FUNCTION_BLOCK CU040AutomatTask EXTENDS CUBaseAutomat IMPLEMENTS ICUTask
VAR

    _missingProcessSettingMessage : TcoCore.TcoMessenger(THIS^);
    _paralellTask : CU040AutomatParalell_1_Task(THIS^, TcoCore.eRestoreMode.None);
	
	//~
    _sb : TcoCore.StringBuilder;
	//~
    _customizedContentInput : CU040DialogContent(THIS^);
END_VAR

VAR
    _dataLoadProcessSettings : BOOL;
    _dataLoadProcessSettingsByPlaner : BOOL;
    _dataCreateNew : BOOL;
    _dataOpen : BOOL;
    _dataClose : BOOL;
    _dataFinalize : BOOL;
    _continueRestore : BOOL;
    _loop : BOOL;
    _inspectionResult : BOOL;
    _inspectionDimensionResult : REAL;
    _tagsPairing : BOOL;
    _reqKey : STRING;
    _reqAssignedValue : STRING;
    _inspectorSingleExamples : BOOL;
    _inspectorGroupExamples : BOOL;
	_dialogExamples : BOOL;

END_VAR

Run();

(*~
	<docu>
		<summary>
			Loads technology settings from the current technology set into this controlled unit.
			The `StationProcessDataManager.Data` is populated by data from process settings.						
		</summary>
	</docu>
~*)
METHOD DataLoadProcessSettings : BOOL
VAR_INPUT
	inStepID : INT;
END_VAR

VAR
	_ans: TcoCore.eDialogAnswer;
END_VAR
IF (Step(inStepID, _dataLoadProcessSettings, 'LOAD PROCESS SETTING')) THEN
    //-------------------------------------
	
	THIS^._missingProcessSettingMessage.OnCondition(Station.Technology.ProcessSettings.Data._EntityId = '')
									   .Build()
									   .Append('No process data. Please load setting')
									   .As()				   
									   .AsError()
									   .Pin();
					   
				   
	IF(Station.Technology.ProcessSettings.Data._EntityId <> '' (*AND NOT THIS^._missingProcessSettingMessage.Pinned*)) THEN
		IF(Station.Technology.ProcessSettings.Read(Station.Technology.ProcessSettings.Data._EntityId).Done) THEN
			Station.ProcessDataManager.Data := Station.Technology.ProcessSettings.Data;
			Station.ProcessDataManager.Data.EntityHeader.RecipeCreated := Station.Technology.ProcessSettings.Data._Created;
			Station.ProcessDataManager.Data.EntityHeader.RecipeLastModified  := Station.Technology.ProcessSettings.Data._Modified;
			Station.ProcessDataManager.Data.EntityHeader.Recipe  := Station.Technology.ProcessSettings.Data._EntityId;				
			CompleteStep();

		END_IF;	
	ELSE
		_ans:=_dialog.Show()
			.WithImage('d:\MTS\Develop\TcOpenGroup\TcOpen\assets\logo\TcOpenWide.png',400,600)	
	       .WithCaption('<#Process data not selected#>')
		   .WithText('<#Would you like to load default settings?#>')
		   .WithYesNoCancel().Answer;
		IF(_ans=TcoCore.eDialogAnswer.Cancel) THEN
			this^.Restore();
		END_IF
		IF( _ans= TcoCore.eDialogAnswer.Yes) THEN
		   
		   	Station.Technology.ProcessSettings.Data._EntityId := 'default';
		END_IF; 

			
	END_IF		    				
    //-------------------------------------
END_IF
END_METHOD

(*~
	<docu>
		<summary>
			Loads process settings from the current process set into this controlled unit.
			The `StationProcessDataManager.Data` is populated by data from process settings.						
		</summary>
	</docu>
~*)
METHOD DataLoadProcessSettingsByPlaner : BOOL
VAR_INPUT
	inStepID : INT;
END_VAR
IF (Step(inStepID, _dataLoadProcessSettingsByPlaner, 'LOAD PROCESS SETTING BY THE PRODUCTION PLANER')) THEN
    //-------------------------------------


								   
	 IF Station.ProductionPlanerTask.Invoke().Done	AND_THEN(Station.ProductionPlanerTask.RequiredProcessSettingsId <> '') THEN
		
		IF NOT Station.ProductionPlanerTask.ProductionPlanCompleted and_then (Station.Technology.ProcessSettings.Read(Station.ProductionPlanerTask.RequiredProcessSettingsId).Done)
			 THEN
			Station.ProcessDataManager.Data := Station.Technology.ProcessSettings.Data;
			Station.ProcessDataManager.Data.EntityHeader.RecipeCreated := Station.Technology.ProcessSettings.Data._Created;
			Station.ProcessDataManager.Data.EntityHeader.RecipeLastModified  := Station.Technology.ProcessSettings.Data._Modified;
			Station.ProcessDataManager.Data.EntityHeader.Recipe  := Station.Technology.ProcessSettings.Data._EntityId;				
			CompleteStep();
			Station.ProductionPlanerTask.Restore();
		END_IF;
	ELSIF  Station.ProductionPlanerTask.ProductionPlanIsEmpty THEN
		IF (_dialog.Show()
	       .WithCaption('<#Production planer#>')
		   .WithText('<#Production planer is empty!#>')
			.WithOk().Answer = TcoCore.eDialogAnswer.OK) THEN;
			;// Production plan comleted , here you can write diferent scenario ( leave it with current state , provide ground etc)	 
	
		 	//Station.GroundTask.Task.Invoke();
		   
		End_if;
	
	ELSIF  Station.ProductionPlanerTask.ProductionPlanCompleted THEN
		IF (_dialog.Show()
	       .WithCaption('<#Production planer#>')
		   .WithText('<#Production planer completed required plan!#>')
			.WithOk().Answer = TcoCore.eDialogAnswer.OK) THEN;
			;// Production plan comleted , here you can write diferent scenario ( leave it with current state , provide ground etc)	 
	
		 	//Station.GroundTask.Task.Invoke();
		   
		End_if;

			
	END_IF		    				
    //-------------------------------------
END_IF
END_METHOD

(*~
	<docu>
		<summary>
			Wait for start operations and then go into this controlled unit sequence.						
		</summary>
	</docu>
~*)
METHOD DataReadyForOperations : BOOL
VAR_INPUT
	inStepID : INT;
END_VAR

VAR
	_ans: TcoCore.eDialogAnswer;
END_VAR
THIS^.Station.ResetReadyForOperations();   

IF (Step(inStepID, TRUE, '<#READY TO START OPERATIONS#>')) THEN
    //-------------------------------------
	
	THIS^.Station.SetReadyForOperations();   
	
  	Await(THIS^.Station.InternalRetrieveEntity(inCarrier:=2(*here comes info from carousel position*),refStorage:=Station.Technology.InternalStorage) 
			 AND_THEN THIS^.Station.DoesBelong() 
			 AND_THEN THIS^.Station.RunOperations(refGlobalTrigger:=Station.Technology.RunOperations)
			 AND_THEN THIS^.Station.InternalOpenEntity(inCarrier:=2(*here comes info from carousel position*),refStorage:=Station.Technology.InternalStorage,inoHeader:= THIS^.Station.CuProcessData.Header));
    //-------------------------------------
END_IF
END_METHOD

METHOD DialogExamples
VAR_INPUT
		inStepID : INT;
END_VAR
IF (Step(inStepID, TRUE, 'DIALOG EXAMPLE ')) THEN
//-------------------------------------
		_dialog.Show()
            .WithType(eDialogType.Question)
            .WithYesNo()
            .WithCaption('Hey')
            .WithText('Do we go ahead ');

        IF (_dialog.Answer = TcoCore.eDialogAnswer.Yes) THEN
            CompleteStep();
        END_IF;

        IF (_dialog.Answer = TcoCore.eDialogAnswer.No) THEN
            ;
        END_IF;

//-------------------------------------
END_IF;

IF (Step(inStepID+10, TRUE, 'DIALOG EXAMPLE WIT IMAGE')) THEN
//-------------------------------------
		_dialog.Show()
            .WithType(eDialogType.Question)
            .WithYesNo()
			.WithImage('D:\MTS\Develop\TcOpenGroup\TcOpen\assets\logo\TcOpenLogo.png',400,600)
            .WithCaption('Hey 1')
            .WithText('Do we go ahead ?');

        IF (_dialog.Answer = TcoCore.eDialogAnswer.Yes) THEN
            CompleteStep();
        END_IF;

        IF (_dialog.Answer = TcoCore.eDialogAnswer.No) THEN
            ;
        END_IF;

//-------------------------------------
END_IF;


IF (Step(inStepID+20, TRUE, 'DIALOG EXAMPLE WITH CLOSE FROM PLC')) THEN
//-------------------------------------
		_dialog.ShowWithExternalClose(inOkAnswerSignal:=FALSE , inYesAnswerSignal:= CurrentStep.Duration>T#2000MS, inNoAnswerSignal:= FALSE, inCancelAnswerSignal:= FALSE)
		    .WithType(eDialogType.Info)
            .WithYesNoCancel()
            .WithCaption('Hey')
            .WithText('Do you wana retry it? Yes answer will be set in 4 sec?');

        IF (_dialog.Answer = TcoCore.eDialogAnswer.Yes) THEN
            CompleteStep();
        END_IF;

      

//-------------------------------------
END_IF;

IF (Step(inStepID+30, TRUE, 'CUSTOMIZED DIALOG EXAMPLE WITH CLOSE FROM PLC ')) THEN
//-------------------------------------
			 _dialogCustomized.ShowWithExternalClose(inOption1AnswerSignal:=FALSE,inOption2AnswerSignal:=FALSE, inOption3AnswerSignal:=CurrentStep.Duration>T#4000MS,inOption4AnswerSignal:=FALSE)
            
            .WithOption1('This is Option1=>retry')
			  .WithOption2('This is Option2=>first step')
			    .WithOption3('This is Option3 =>continue and finish in 4s')
			.WithImage('D:\MTS\Develop\TcOpenGroup\TcOpen\assets\logo\TcOpenWide.png',500,500)
            .WithCaption('Hey')
            .WithText('What we are going to do.');
            
		
           
	
			IF (_dialogCustomized.Answer = TcoCore.eCustomizedDialogAnswer.Option3) THEN
				CompleteStep();
			END_IF;

//-------------------------------------
END_IF;

IF (Step(inStepID+40, TRUE, 'INPUT DIALOG EXAMPLE  REQURED FIELDS TO INPUT DATA')) THEN
//-------------------------------------
		_dialogWithInput.Show(refContent:=_customizedContentInput)
            .WithType(eDialogType.Question)
            .WithYesNo()
            .WithCaption('Hey wana set data')
            .WithText('Do you realy want to sent data to ....?');
                
		IF (_dialogWithInput.Answer = TcoCore.eInputDialogAnswer.Yes) THEN
				CompleteStep();
			//by yes or (ok) option data are confirmed and transfered to plc (_customizedContentInput)
		ELSIF (_dialogWithInput.Answer = TcoCore.eInputDialogAnswer.No) THEN
			// data in struct '_customizedContentInput' remains same as before
 		END_IF;
		

//-------------------------------------
END_IF;
IF (Step(inStepID+50, TRUE, 'INPUT DIALOG EXAMPLE WITH WEB CONTENT AND REQURED FIELDS TO INPUT DATA')) THEN
//-------------------------------------
		_dialogWithInput.Show(refContent:=_customizedContentInput)
            .WithType(eDialogType.Question)
            .WithOk()
			.WithImage('https://github.com/TcOpenGroup',400,600)
            .WithCaption('Hey wana set data')
            .WithText('Do you realy want to sent data to ....?');
			
                
		IF (_dialogWithInput.Answer = TcoCore.eInputDialogAnswer.OK) THEN
			CompleteStep();
			
		END_IF;

//-------------------------------------
END_IF;
END_METHOD

METHOD GroupedExample
VAR_INPUT
		inStepID : INT;
END_VAR
IF (Step(inStepID, TRUE, 'MULTI ANALOGUE INSPECTIONS PART 1 WITH WEB CONTENT')) THEN
//-------------------------------------
		Station.GroupInspection
		.WithCoordinator(THIS^)
		.Act();
		Station.GroupInspection.Inspect(Station.ProcessDataManager.Data.CU040.Dim_Inspector_1.WithCoordinator(THIS^).Inspect(0));	
		Station.GroupInspection.Inspect(Station.ProcessDataManager.Data.CU040.Dim_Inspector_2.WithCoordinator(THIS^).Inspect(0));	
		Station.GroupInspection.Inspect(Station.ProcessDataManager.Data.CU040.Dim_Inspector_3.WithCoordinator(THIS^).Inspect(0));	
		Station.GroupInspection.Inspect(Station.ProcessDataManager.Data.CU040.Dim_Inspector_4.WithCoordinator(THIS^).Inspect(0));	
		Station.GroupInspection.Inspect(Station.ProcessDataManager.Data.CU040.Dim_Inspector_5.WithCoordinator(THIS^).Inspect(0));	
		Station.GroupInspection.Inspect(Station.ProcessDataManager.Data.CU040.Dim_Inspector_6.WithCoordinator(THIS^).Inspect(1));	
		Station.GroupInspection.Inspect(Station.ProcessDataManager.Data.CU040.Dim_Inspector_7.WithCoordinator(THIS^).Inspect(0));	
		Station.GroupInspection.Inspect(Station.ProcessDataManager.Data.CU040.Dim_Inspector_8.WithCoordinator(THIS^).Inspect(0));	
		Station.GroupInspection.Inspect(Station.ProcessDataManager.Data.CU040.Dim_Inspector_9.WithCoordinator(THIS^).Inspect(0));	
		Station.GroupInspection.Inspect(Station.ProcessDataManager.Data.CU040.Dim_Inspector_10.WithCoordinator(THIS^).Inspect(0));	
	
		
		Station.GroupInspection.UpdateComprehensiveResult(Station.ProcessDataManager.Data.EntityHeader.Results)	
		.Instruct('Something is wrong 1')
		.InstructWithImage('https://github.com/TcOpenGroup/TcOpen/blob/dev/README.md',400,600)	
		.OnFail()
		.Dialog(inStepID+10);			
//-------------------------------------
END_IF;

IF (Step(inStepID+10, TRUE, 'MULTI ANALOGUE INSPECTIONS PART 2 WITH INSTRUCTION AND DESCRIPTION')) THEN
//-------------------------------------
		Station.GroupInspection
		.WithCoordinator(THIS^)
		.Act();
		Station.GroupInspection.Inspect(Station.ProcessDataManager.Data.CU040.Dim_Inspector_11.WithCoordinator(THIS^).Inspect(0));	
		Station.GroupInspection.Inspect(Station.ProcessDataManager.Data.CU040.Dim_Inspector_12.WithCoordinator(THIS^).Inspect(0));	
		Station.GroupInspection.Inspect(Station.ProcessDataManager.Data.CU040.Dim_Inspector_13.WithCoordinator(THIS^).Inspect(0));	
		Station.GroupInspection.Inspect(Station.ProcessDataManager.Data.CU040.Dim_Inspector_14.WithCoordinator(THIS^).Inspect(0));	
		Station.GroupInspection.Inspect(Station.ProcessDataManager.Data.CU040.Dim_Inspector_15.WithCoordinator(THIS^).Inspect(0));	
		Station.GroupInspection.Inspect(Station.ProcessDataManager.Data.CU040.Dim_Inspector_16.WithCoordinator(THIS^).Inspect(1));	
		Station.GroupInspection.Inspect(Station.ProcessDataManager.Data.CU040.Dim_Inspector_17.WithCoordinator(THIS^).Inspect(0));	
		Station.GroupInspection.Inspect(Station.ProcessDataManager.Data.CU040.Dim_Inspector_18.WithCoordinator(THIS^).Inspect(0));	
		Station.GroupInspection.Inspect(Station.ProcessDataManager.Data.CU040.Dim_Inspector_19.WithCoordinator(THIS^).Inspect(0));	
		Station.GroupInspection.Inspect(Station.ProcessDataManager.Data.CU040.Dim_Inspector_20.WithCoordinator(THIS^).Inspect(0));	
	
		
		Station.GroupInspection.UpdateComprehensiveResult(Station.ProcessDataManager.Data.EntityHeader.Results)	
		.WithDescription()
		.Instruct('Something is wrong 2')
		.OnFail()
		.Dialog(inStepID+20);			
//-------------------------------------
END_IF;



IF (Step(inStepID+20, TRUE, 'MULTI ANALOGUE INSPECTIONS PART 2 WITH INSTRUCTION AND DESCRIPTION EVAVLUATED')) THEN
//-------------------------------------

		Station.GroupInspection
		.WithCoordinator(THIS^)
		.Act();
		Station.GroupInspection.Inspect(Station.ProcessDataManager.Data.CU040.Dim_Inspector_11.WithCoordinator(THIS^).Inspect(0));	
		Station.GroupInspection.Inspect(Station.ProcessDataManager.Data.CU040.Dim_Inspector_12.WithCoordinator(THIS^).Inspect(0));	
		Station.GroupInspection.Inspect(Station.ProcessDataManager.Data.CU040.Dim_Inspector_13.WithCoordinator(THIS^).Inspect(0));	
		Station.GroupInspection.Inspect(Station.ProcessDataManager.Data.CU040.Dim_Inspector_14.WithCoordinator(THIS^).Inspect(0));	
		Station.GroupInspection.Inspect(Station.ProcessDataManager.Data.CU040.Dim_Inspector_15.WithCoordinator(THIS^).Inspect(0));	
		Station.GroupInspection.Inspect(Station.ProcessDataManager.Data.CU040.Dim_Inspector_16.WithCoordinator(THIS^).Inspect(1));	
		Station.GroupInspection.Inspect(Station.ProcessDataManager.Data.CU040.Dim_Inspector_17.WithCoordinator(THIS^).Inspect(0));	
		Station.GroupInspection.Inspect(Station.ProcessDataManager.Data.CU040.Dim_Inspector_18.WithCoordinator(THIS^).Inspect(0));	
		Station.GroupInspection.Inspect(Station.ProcessDataManager.Data.CU040.Dim_Inspector_19.WithCoordinator(THIS^).Inspect(0));	
		Station.GroupInspection.Inspect(Station.ProcessDataManager.Data.CU040.Dim_Inspector_20.WithCoordinator(THIS^).Inspect(0));	
	
		
		Station.GroupInspection.UpdateComprehensiveResult(Station.ProcessDataManager.Data.EntityHeader.Results)	
		.WithDescription()
		.Instruct('Something is wrong')
		.OnFail().Evaluate(	inStepID+10,eTcoInspectorFailMode.RetryThenCarryOn,inStepId+30);
//-------------------------------------
END_IF;

IF (Step(inStepID+30, TRUE, 'DONE')) THEN
//-------------------------------------
		CompleteStep();
//-------------------------------------
END_IF;
END_METHOD

(*~
	<docu>
		<summary>
			Main method of the sequener. Custom code needs to be placed here. The sequencer is executed by call of **Instance.Run()** method.
			This method is abstract, and it must be overridden in derived block.
		</summary>
	</docu>
~*)
METHOD PROTECTED Main : BOOL
(*

	OPENING DATA OPERATIONS
	Following methods provide process data manipulation for this controlled unit.
	Remove `IF` statement and comment or uncomment according to your need.
*)
// Loads process settings. 
// Typically used in the first station of the technology to load process settings that will be used trough out the production
IF (_dataLoadProcessSettings) THEN
    THIS^.DataLoadProcessSettings(100);
END_IF;

// Loads process settings via produciton planer. 
// Typically used in the first station of the technology to load process settings that will be used trough out the production 
// .......
IF (_dataLoadProcessSettingsByPlaner) THEN
    THIS^.DataLoadProcessSettingsByPlaner(110);
END_IF;

(*

		
		This step we would like to star cycle time (e.g. we want to exclude loading data from clean cycle time )		
*)
IF (Step(150, TRUE, '<#START MEASURE CT TRIGGER#>')) THEN
    //-------------------------------------    
    StartCleanCycleTime();

	CustomObserver.DefineControledUnit(THIS^.Station.CuId);
	
    StepCompleteWhen(TRUE);
    //-------------------------------------
END_IF

// Creates new data entity (new part/item) 
// Typically used in the first station of the technology to create new document/record to be persited in the repository.
// Sets the status of the entity to 'InProgress'
IF (_dataCreateNew) THEN
	IF (Step(160, TRUE, 'CREATE ENTIY ID')) THEN
		//-------------------------------------    
		Station.ProcessDataManager.Data._EntityId := ULINT_TO_STRING(Context.RealTimeClock.TickClock());
	
		StepCompleteWhen(Station.ProcessDataManager.Data._EntityId<>'');
		//-------------------------------------
	END_IF
    THIS^.DataEntityCreateNew(200, Station.ProcessDataManager.Data._EntityId, Header := Station.ProcessDataManager.Data.CU040.Header);
END_IF;

// Populates the information in the data header of this controlled unit (operation start time stamp, user info, etc)
// Typically used prior to starting operation within a controlled unit.
IF (_dataOpen) THEN
    THIS^.DataEntityOpen(300,
        30000,
        Station.ProcessDataManager.Data._EntityId,
        Station.ProcessDataManager.Data.CU040.Header);
END_IF;


// Handle user defined carier id
// Typically used in the first station of the technology to assign user defined carier ID  instead of raw unique id(RfidChip....)
IF (_tagsPairing) THEN
    THIS^.PairTag(400);
END_IF;
(*

		STEPS OF THE SEQUENCE
		Here we would place steps to perfom the operations of this controlled unit.

*)



IF (Step(900, TRUE, 'SINGLE INSPECTION')) THEN
    //-------------------------------------    
	Station.ProcessDataManager.Data.CU040.BoltPresenceInspector.Data.FailureDescription:='BoltPresenceInspector error';
    Station.ProcessDataManager.Data.CU040.BoltPresenceInspector.WithCoordinator(THIS^)
        .Inspect(_inspectionResult)
        .UpdateComprehensiveResult(Station.ProcessDataManager.Data.EntityHeader.Results)
        .OnFail().CarryOn();
    //-------------------------------------
END_IF

IF (Step(910, TRUE, 'SINGLE ANALOGUE INSPECTION')) THEN
    //-------------------------------------    
		Station.ProcessDataManager.Data.CU040.BoltDimensionPresenceInspector.Data.FailureDescription:='BoltDimensionPresenceInspector error';

    Station.ProcessDataManager.Data.CU040.BoltDimensionPresenceInspector.WithCoordinator(THIS^)
        .Inspect(_inspectionDimensionResult)
        .UpdateComprehensiveResult(Station.ProcessDataManager.Data.EntityHeader.Results)
        .OnFail().Dialog(300);
    //-------------------------------------
END_IF


//dialog usage examples
IF _dialogExamples THEN
	DialogExamples(1000);
END_IF;

//single inspexction usage
IF _inspectorSingleExamples THEN
	SingleExample(1100);
END_IF;

// grouped usage of isnpectors
IF _inspectorGroupExamples THEN
	GroupedExample(1200);
END_IF;


IF (Step(2000, true, 'START PARALELL TASK')) THEN
    //-------------------------------------    
    StepCompleteWhen(_paralellTask.Task.Invoke().Busy);
    //-------------------------------------
END_IF

(*

		RECOVERY STEPS
		This step and the following steps should bring the controlled unit in a state from which 
		the sequence can be safely restarted from the beginning of the this sequencer. 		
*)
IF (Step(RESTORE_STEP_ID, TRUE, 'FIRST RESTORE STEP')) THEN
    //-------------------------------------
    StepCompleteWhen(_continueRestore);
    //-------------------------------------	
END_IF

(*

		
		This step we would save cycle time value (e.g. we not include saving data into cycle time )
		
*)
IF (Step(2150, TRUE, 'STOP MEASURE CT TRIGGER')) THEN
    //-------------------------------------    
    StopCleanCycleTime();
    StepCompleteWhen(TRUE);
    //-------------------------------------
END_IF

(*

	CLOSING DATA OPERATIONS
	Following methods provide process data manipulation for this controlled unit.
	Comment or uncomment according to your need.
*)
// Populates the information in the data header of this controlled unit (operations end time stamp, user info, etc)
// Typically used after all steps within the controlled unit are completed.
IF (_dataClose) THEN
    THIS^.DataEntityClose(5000, eDataEntityInvokeType.InvokeAndWaitDone, Station.ProcessDataManager.Data.CU040.Header);
END_IF;

// Populates the information in the data header of this controlled unit (operations end time stamp, user info, etc)
// Typically used after all operation on the technology are completed.
// Input parameter eDataEntityInvokeType.InvokeOnly is used for speed up cycle(TRUE)
IF (_dataFinalize) THEN
    THIS^.DataEntityFinalize(5500, eDataEntityInvokeType.InvokeOnly, Station.ProcessDataManager.Data.CU040.Header);
END_IF;

IF (Step(10000, TRUE, 'WAIT FOR PARALELL TASK TO FINISH')) THEN
    //-------------------------------------
    StepCompleteWhen(_paralellTask.Task.Done);

    IF _paralellTask.Task.Done THEN
        _paralellTask.Restore();
		
    END_IF
    //-------------------------------------	
END_IF

IF (Step(20000, _dataClose, 'WAIT FOR IF DATA FINALIZE IS DONE')) THEN
    //-------------------------------------
    StepCompleteWhen(Station.UpdateEntityTask.Done);
	CustomObserver.SetCycleId(Station.ProcessDataManager.Data._EntityId);
    //-------------------------------------	
END_IF



//monitor if conseccutive failures occur during automatic cycle. System monitor two basic types like are arbitrary failure in seqence, or  same(equal) failure in sequence
//if Number of allowed recurring failure is 0 , monitoring is inactive.
//Recurring failures are based on ErrorCodes in TcoComprehensiveResult.
//If error code in Same recurring failure is empty string ,monitorig of failure is not performed.
//Error code in Arbitrary Recuring failure is irelevant.    
THIS^.MonitorAnyRecurringFailure(22000,THIS^.Station._settings.AnyRecurringFailure>0 , Station.ProcessDataManager.Data.EntityHeader.Results);
THIS^.MonitorSameRecurringFailure(22100,THIS^.Station._settings.SameRecurringFailure>0 , Station.ProcessDataManager.Data.EntityHeader.Results);



IF (Step(30000, TRUE, 'LAST STEP')) THEN
    //-------------------------------------

		IF (_loop) THEN
			CompleteSequence();
		END_IF;


    //-------------------------------------	
END_IF

_paralellTask();
END_METHOD

METHOD PUBLIC OnStart
SUPER^.OnStart();
Station.GroundTask.Restore();
Station.ManualTask.Restore();
Station.GroundTask.CancelGround();
_paralellTask.Restore();
END_METHOD

(*~
	<docu>
		<summary>
			Loads process settings from the current process set into this controlled unit.
			The `StationProcessDataManager.Data` is populated by data from process settings.						
		</summary>
	</docu>
~*)
METHOD PairTag : BOOL
VAR_INPUT
	inStepID : INT;
END_VAR

VAR
	answer: TagsPairing;
	_addNewTag: BOOL;
	dialogAnswer: eDialogAnswer;
END_VAR
IF (Step(inStepID, _tagsPairing, '<#PAIR TAG WITH ASSIGNED VALUE EXAMPLE#>')) THEN
    //-------------------------------------
	_addNewTag:=FALSE;

	answer:= Station.Components.PairTagTask.Answer;
	//this field may be assigned by unique ID of rfid chip , or dmc code.The PairTagTask provide answer where is assigned user defined value for this unique ID value.
	//If not, there may be diferent scenarios defined. See example bellow.
	_reqKey:='123456789';				   
	 IF Station.Components.PairTagTask.Run(inMode:=eTagPairingMode.GetTag, inKey:=_reqKey ,inAssignedValue:='').Invoke().Done	 THEN
		
		IF  answer.Answer =eTagPairingAnswer.TagFound 
			 THEN
			Station.ProcessDataManager.Data.EntityHeader.Carrier := answer.AssignedValue;
			CompleteStep();
			Station.Components.PairTagTask.Restore();
		
		ELSIF  answer.Answer = eTagPairingAnswer.TagFoundInactive THEN
			IF (_dialog.Show()
			   .WithCaption('<#Pairing Tag#>')
			   .WithText(_sb.Clear().Append('<#Founded tag#> ').Append(_reqKey).Append(' <#is inactive!#> ').Append(Station.Components.PairTagTask.AnswerInstruction).ToString() )
				.WithOk().Answer = TcoCore.eDialogAnswer.OK) THEN;
				;// Founded tag is Inactive. Probably carier(pallete) was disasbled due produced many errors.Se  here you can write diferent scenario ( leave it with current state , provide ground etc)	 
		
				//Station.GroundTask.Task.Invoke();
			   
			End_if;
		
		ELSIF  answer.Answer = eTagPairingAnswer.TagFoundAssignedValueEmpty THEN
			  IF (_dialog.Show()
			   .WithCaption('<#Pairing Tag#>')
			   .WithText(_sb.Clear().Append('<#Tag#> ').Append(_reqKey).Append(' <#is founded but assigned value is empty! Would you like continue?#> ').Append(Station.Components.PairTagTask.AnswerInstruction).ToString() )
				.WithYesNo().Answer = TcoCore.eDialogAnswer.Yes) THEN;
				CompleteStep();
				Station.Components.PairTagTask.Restore();
			END_IF;
		   
		ELSIF  answer.Answer = eTagPairingAnswer.TagNotFound THEN
			  IF (_dialog.Show()
			   .WithCaption('<#Pairing Tag#>')
			   .WithText(_sb.Clear().Append('<#Tag#> ').Append(_reqKey).Append(' <#is not founded ! Would you like assign right now?#> ').Append(Station.Components.PairTagTask.AnswerInstruction).ToString() )
				.WithYesNo().Answer = TcoCore.eDialogAnswer.Yes) THEN;
				_addNewTag:=TRUE;
				CompleteStep();
				Station.Components.PairTagTask.Restore();
			END_IF;
	
		
			ELSIF  answer.Answer = eTagPairingAnswer.EmptyCollection THEN
			  IF (_dialog.Show()
			   .WithCaption('<#Pairing Tag#>')
			   .WithText(_sb.Clear().Append('<#Tag#> ').Append(_reqKey).Append(' <#is not founded due collection is empty ! Would you like assign right now?#> ').Append(Station.Components.PairTagTask.AnswerInstruction).ToString() )
				.WithYesNo().Answer = TcoCore.eDialogAnswer.Yes) THEN;
				_addNewTag:=TRUE;
				CompleteStep();
				Station.Components.PairTagTask.Restore();
			END_IF;
		End_if;
			
	END_IF		    				
    //-------------------------------------
END_IF

IF (Step(inStepID+10, _tagsPairing AND _addNewTag, '<#ADD NEW TAG  EXAMPLE#>')) THEN
    //-------------------------------------
	
	answer:= Station.Components.PairTagTask.Answer;
	//this field may be assigned by unique ID of rfid chip , or dmc code.The PairTagTask provide answer where is assigned user defined value for this unique ID value.
	//If not, there may be diferent scenarios defined. See example bellow.
	_reqKey:='123456789';		
	_reqAssignedValue := 'CustomIdExample123';	   
	 IF Station.Components.PairTagTask.Run(inMode:=eTagPairingMode.AddTag, inKey:=_reqKey, inAssignedValue:=_reqAssignedValue).Invoke().Done	 THEN
		
		IF  answer.Answer =eTagPairingAnswer.TagAddedSuccessfully 
			 THEN
			Station.ProcessDataManager.Data.EntityHeader.Carrier := answer.AssignedValue;
			CompleteStep();
			Station.Components.PairTagTask.Restore();
		END_IF;
	ELSIF  answer.Answer = eTagPairingAnswer.TagAlreadyExist THEN
		IF (_dialog.Show()
	       .WithCaption('<#Adding Tag#>')
		   .WithText(_sb.Clear().Append('<#Tag#> ').Append(_reqKey).Append(' <#already exist!#> ').Append(Station.Components.PairTagTask.AnswerInstruction).ToString() )
			.WithOk().Answer = TcoCore.eDialogAnswer.OK) THEN;
			;// Founded tag is Inactive. Probably carier(pallete) was disasbled due produced many errors.Se  here you can write diferent scenario ( leave it with current state , provide ground etc)	 
	
		 	//Station.GroundTask.Task.Invoke();
		   
		End_if;
	
	ELSIF  answer.Answer = eTagPairingAnswer.TagAddedNotSuccessfuly THEN
			dialogAnswer := _dialog.Show()
	       .WithCaption('<#Pairing Tag#>')
		   .WithText(_sb.Clear().Append('<#Tag#> ').Append(_reqKey).Append(' <#was not founnd! Would you like still like to continue?#> ').Append(Station.Components.PairTagTask.AnswerInstruction).ToString() )
			.WithYesNo().Answer;
			
	      IF (dialogAnswer= TcoCore.eDialogAnswer.Yes) THEN;
			CompleteStep();
			Station.Components.PairTagTask.Restore();
		END_IF;
		   

			
	END_IF		    				
    //-------------------------------------
END_IF
END_METHOD

METHOD SingleExample : BOOL
VAR_INPUT
		inStepID : INT;
END_VAR

IF (Step(inStepID, TRUE, 'SINGLE INSPECTION')) THEN
    //-------------------------------------    
	Station.ProcessDataManager.Data.CU040.BoltPresenceInspector.Data.FailureDescription:='BoltPresenceInspector error';
    Station.ProcessDataManager.Data.CU040.BoltPresenceInspector.WithCoordinator(THIS^)
        .Inspect(_inspectionResult)
        .UpdateComprehensiveResult(Station.ProcessDataManager.Data.EntityHeader.Results)
        .OnFail().Dialog(inStepID+10);
    //-------------------------------------
END_IF

// with checking if specific inspector is overinspected
IF (Step(inStepID+10, TRUE, 'SINGLE ANALOGUE INSPECTION')) THEN
//-------------------------------------
	Station.ProcessDataManager.Data.CU040.BoltDimensionPresenceInspector.Data.FailureDescription:='BoltDimensionPresenceInspector error';
	Station.ProcessDataManager.Data.CU040.BoltDimensionPresenceInspector.Data.NumberOfAllowedRetries:=100;
	IF NOT Station.ProcessDataManager.Data.CU040.BoltDimensionPresenceInspector.OverInspected THEN
	
		Station.ProcessDataManager.Data.CU040.BoltDimensionPresenceInspector.WithCoordinator(THIS^)
			.Inspect(_inspectionDimensionResult)
			.WithDescription()
			.UpdateComprehensiveResult(Station.ProcessDataManager.Data.EntityHeader.Results)
			.OnFail().Retry(inStepID+20);
	ELSE
	 	RequestStep(RESTORE_STEP_ID);	
	END_IF
//-------------------------------------
END_IF;

IF (Step(inStepID+20, TRUE, 'DONE')) THEN
//-------------------------------------
		CompleteStep();
//-------------------------------------
END_IF;
END_METHOD

PROPERTY Station : REFERENCE TO CU040
GET
VAR
    _station : POINTER TO CU040;
END_VAR
IF __QUERYPOINTER(Parent, _station) THEN // Check if _Parent is Station001
    Station REF= _station^;              // If the check is successful dereference a pointer. simlar to THIS^ or SUPER^
END_IF
END_GET
END_PROPERTY

END_FUNCTION_BLOCK

(* stored: Version 1.1.0.1
   POU CU040AutomatTask: Id {2f93a84b-96c3-4767-9354-8489dc257b5f}, SpecialFunc None
   Folder DataOperations: Id {8c5e9a2b-e87a-408f-8006-7110103ad605}
   Folder InpspectorExamples: Id {ab0428cf-f046-4c16-bd60-c715f03f0c0a}
   Folder ProductionPlaner: Id {ba187764-f90f-4d21-9fa4-3797e7025e59}
   Folder TagsPairing: Id {cc57f27d-65a9-48eb-8cfe-c83a814b9eff}
   Method DataLoadProcessSettings: Id {48d24ce4-215a-4d7a-a4bd-38a0b814bc66}
   Method DataLoadProcessSettingsByPlaner: Id {daf574f2-b3b5-403f-96a9-568008259533}
   Method DataReadyForOperations: Id {4563f6f9-e2a1-4b24-94c1-fceb5ce9ad36}
   Method DialogExamples: Id {b7b9fc9e-a0e6-4d47-b1c4-7595df40910a}
   Method GroupedExample: Id {eb1ca8d3-6d95-4b44-8595-95d56c35566e}
   Method Main: Id {8adbac45-28c1-43da-bc61-1fc46bc78461}
   Method OnStart: Id {1745381b-75a6-4c5b-8ae6-0b2dfcbd36e2}
   Method PairTag: Id {e2e7e616-86ca-438b-9908-f256660671fc}
   Method SingleExample: Id {24dc60c3-501d-496e-8d24-3b5ad4594612}
   Property Station: Id {02782738-b1b9-4083-87bb-5f1b248eccf1}
   Get Get: Id {e7c8a954-4a55-4917-878a-321178a40bd7} *)
